FUNCTION BytesToUInt16 : UINT

VAR_INPUT
  highByte : BYTE;  // Most‐significant byte
  lowByte  : BYTE;  // Least‐significant byte
END_VAR

VAR
  _hb  : UINT;
  _lb  : UINT;
END_VAR


// Shift the high byte into bits 8–15, then OR in the low byte
_hb := SHL( TO_UINT(highByte), 8 );
_lb := TO_UINT(lowByte);
BytesToUInt16 := _hb OR _lb;

END_FUNCTION

(* stored: Version 1.1.0.1
   POU BytesToUInt16: Id {92b8578c-be43-415e-9d8c-b36e682fd1ad}, SpecialFunc None *)
